PROGRAM PRG_IM5K4_PPM
VAR
    {attribute 'pytmc' := '
        pv: IM5K4:PPM
        io: io
    '}
    {attribute 'TcLinkTo' := '.fbGige.iIlluminatorINT 					:= TIIB[IM5K4-EL4004-E7]^AO Outputs Channel 1^Analog output;
                              .fbGige.bGigePower 						:= TIIB[IM5K4-EL2004-E3]^Channel 2^Output;
                              .fbPowerMeter.iVoltageINT 				:= TIIB[IM5K4-EL3062-E6]^AI Standard Channel 1^Value;
                              .fbPowerMeter.fbThermoCouple.bError 		:= TIIB[IM5K4-EL3314-E4]^TC Inputs Channel 1^Status^Error;
                              .fbPowerMeter.fbThermoCouple.bUnderrange	:= TIIB[IM5K4-EL3314-E4]^TC Inputs Channel 1^Status^Underrange;
                              .fbPowerMeter.fbThermoCouple.bOverrange 	:= TIIB[IM5K4-EL3314-E4]^TC Inputs Channel 1^Status^Overrange;
                              .fbPowerMeter.fbThermoCouple.iRaw 		:= TIIB[IM5K4-EL3314-E4]^TC Inputs Channel 1^Value;
                              .fbYagThermoCouple.bError 				:= TIIB[IM5K4-EL3314-E4]^TC Inputs Channel 2^Status^Error;
                              .fbYagThermoCouple.bUnderrange 			:= TIIB[IM5K4-EL3314-E4]^TC Inputs Channel 2^Status^Underrange;
                              .fbYagThermoCouple.bOverrange 			:= TIIB[IM5K4-EL3314-E4]^TC Inputs Channel 2^Status^Overrange;
                              .fbYagThermoCouple.iRaw 					:= TIIB[IM5K4-EL3314-E4]^TC Inputs Channel 2^Value'}
    fbIM5K4: FB_PPM;
    fStartupVelo: LREAL := 12;

    {attribute 'TcLinkTo' := '.iRaw 					:= TIIB[IM5K4-EL3052-E5]^AI Standard Channel 1^Value; '}
    fbFDQTest : FB_AnalogInput;

END_VAR



fbIM5K4.stOut.fPosition := -5.13;
fbIM5K4.stOut.fVelocity := fStartupVelo;
fbIM5K4.stOut.bUseRawCounts := FALSE;
fbIM5K4.stOut.bValid := TRUE;
fbIM5K4.stOut.stPMPS.sPmpsState := 'IM5K4:PPM-OUT';

fbIM5K4.stPower.fPosition := -44.23;
fbIM5K4.stPower.fVelocity := fStartupVelo;
fbIM5K4.stPower.bUseRawCounts := FALSE;
fbIM5K4.stPower.bValid := TRUE;
fbIM5K4.stPower.stPMPS.sPmpsState := 'IM5K4:PPM-POWERMETER';

fbIM5K4.stYag1.fPosition := -68.23;
fbIM5K4.stYag1.fVelocity := fStartupVelo;
fbIM5K4.stYag1.bUseRawCounts := FALSE;
fbIM5K4.stYag1.bValid := TRUE;
fbIM5K4.stYag1.stPMPS.sPmpsState := 'IM5K4:PPM-YAG1';

fbIM5K4.stYag2.fPosition := -94.24;
fbIM5K4.stYag2.fVelocity := fStartupVelo;
fbIM5K4.stYag2.bUseRawCounts := FALSE;
fbIM5K4.stYag2.bValid := TRUE;
fbIM5K4.stYag2.stPMPS.sPmpsState := 'IM5K4:PPM-YAG2';

fbIM5K4(
    fbArbiter := fbArbiter,
    fbFFHWO := fbFastFaultOutput1,
    stYStage := Main.M17,
    sPmpsDeviceName := 'IM5K4:PPM',
    sTransitionKey := 'IM5K4:PPM-TRANSITION',

);

fbFDQtest(iTermBits:=12, fTermMax:=60, fTermMin:=0);

END_PROGRAM

(* stored: Version 1.1.0.1, ProductVersion 3.1.4022.18
   POU PRG_IM5K4_PPM: Id {70ab2a3c-97c1-4d17-a072-939f2529a358}, SpecialFunc None *)
